// TIA Portal V21 export
// export: Created 2026-08-11T14:59:46Z, ExportSetting WithDefaults
VAR_GLOBAL   // PLC tag table "AnalogOutputs"
   Outfeed_Speed AT %QW64 : Int;   // Outfeed conveyor drive - speed reference
END_VAR
